// TIA Portal V20 export
FUNCTION_BLOCK "LER_hotPressLeftHistory"   // FB75, LAD
// stored: Access Published, MemoryReserve 100, SetENOAutomatically false
   VAR_INPUT
      finished : Bool;
      partID : String[32];
      ProductionTimestamp : DTL;
      result : Bool;
   END_VAR
   VAR_IN_OUT
      dataLog : "LER_typeServoPressHistory";
   END_VAR
   VAR
      statDataLogDelete { S7_SetPoint := 'True'} : "LER_typeServoPressHistory";
      statHold { S7_SetPoint := 'True'} : Bool;
      statExecute { S7_SetPoint := 'True'} : Bool;
      statMoveDone : Bool;
      statComplete { S7_SetPoint := 'True'} : Bool;
   END_VAR
   VAR_TEMP
      tempRetVal : Array[0..9] of Int;
      tempTrigger : Bool;
   END_VAR
   VAR_TEMP   // added for the SCL form of the ladder/FBD networks
      _w1 : Bool;
   END_VAR
BEGIN

REGION Network 1
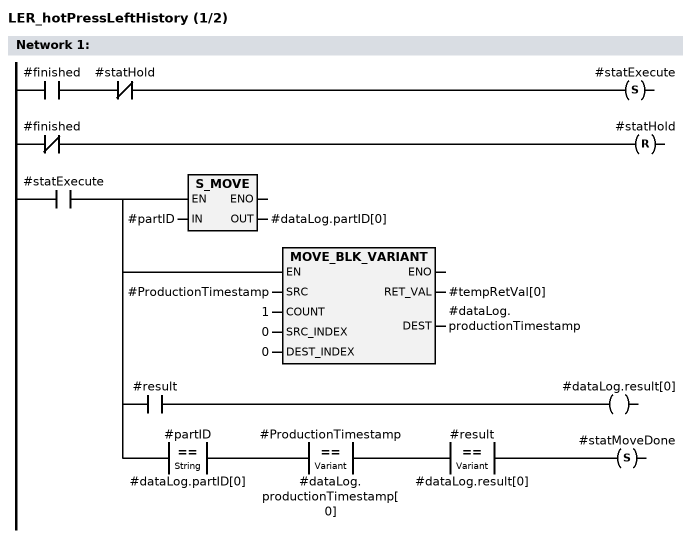
   RUNG wire#powerrail
      Contact( #finished )
      I_Contact( #statHold )
      S_Coil( #statExecute )
   END_RUNG
   RUNG wire#powerrail
      I_Contact( #finished )
      R_Coil( #statHold )
   END_RUNG
   RUNG wire#powerrail
      Contact( #statExecute )
      wire#w1
      S_Move(in := #partID, out => #dataLog.partID[0])
   END_RUNG
   RUNG wire#w1
      MOVE_BLK_VARIANT(SRC := #ProductionTimestamp, COUNT := 1, SRC_INDEX := 0, DEST_INDEX := 0, Ret_Val => #tempRetVal[0], DEST => #dataLog.productionTimestamp)
   END_RUNG
   RUNG wire#w1
      Contact( #result )
      Coil( #dataLog.result[0] )
   END_RUNG
   RUNG wire#w1
      { S7_Templates := "SrcType := String" } EQ_Contact(in1 := #partID, in2 := #dataLog.partID[0])
      { S7_Templates := "SrcType := Variant" } EQ_Contact(in1 := #ProductionTimestamp, in2 := #dataLog.productionTimestamp[0])
      { S7_Templates := "SrcType := Variant" } EQ_Contact(in1 := #result, in2 := #dataLog.result[0])
      S_Coil( #statMoveDone )
   END_RUNG
   // the same network as SCL:
   IF #finished AND NOT #statHold THEN #statExecute := TRUE; END_IF;
   IF NOT #finished THEN #statHold := FALSE; END_IF;
   IF #statExecute THEN
       #dataLog.partID[0] := #partID;
       #tempRetVal[0] := MOVE_BLK_VARIANT(SRC := #ProductionTimestamp,
                               COUNT := 1,
                               SRC_INDEX := 0,
                               DEST_INDEX := 0,
                               DEST => #dataLog.productionTimestamp);
   END_IF;
   #dataLog.result[0] := #statExecute AND #result;
   IF #statExecute AND (#partID = #dataLog.partID[0]) AND (#ProductionTimestamp = #dataLog.productionTimestamp[0]) AND (#result = #dataLog.result[0]) THEN
       #statMoveDone := TRUE;
   END_IF;
END_REGION

REGION Network 2
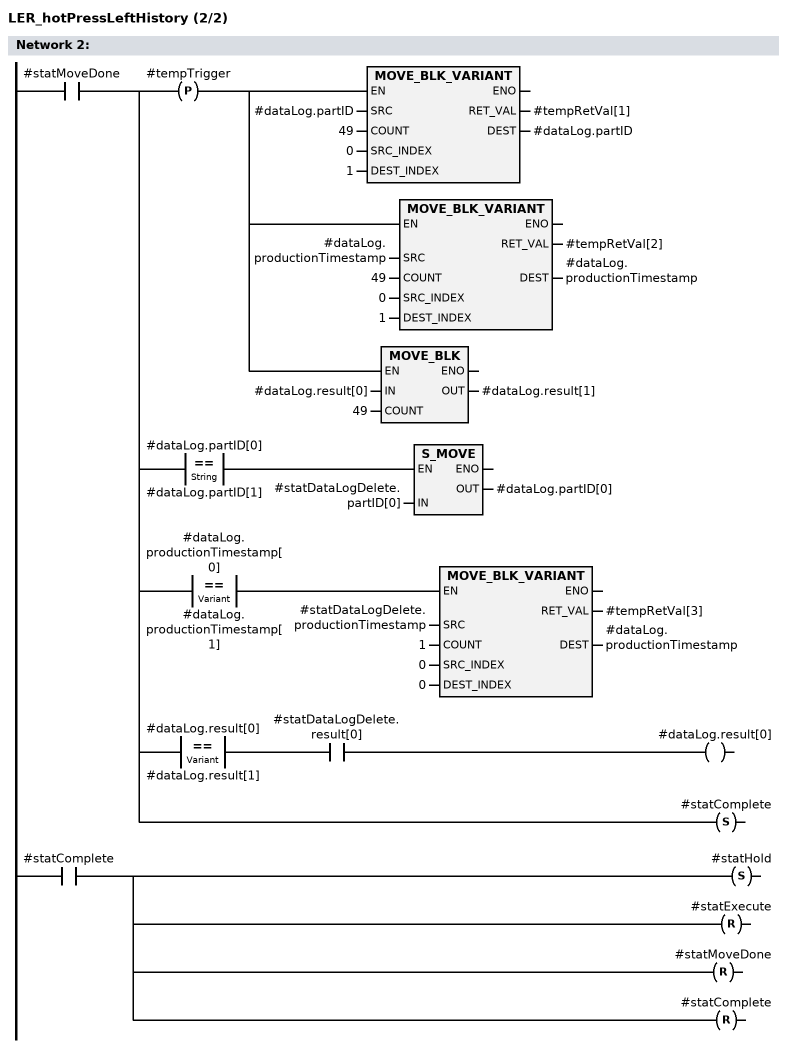
   #_w1 := #statMoveDone AND NOT #tempTrigger;   // rising edge
   #tempTrigger := #statMoveDone;
   IF #_w1 THEN
       #tempRetVal[1] := MOVE_BLK_VARIANT(SRC := #dataLog.partID,
                               COUNT := 49,
                               SRC_INDEX := 0,
                               DEST_INDEX := 1,
                               DEST => #dataLog.partID);
       #tempRetVal[2] := MOVE_BLK_VARIANT(SRC := #dataLog.productionTimestamp,
                               COUNT := 49,
                               SRC_INDEX := 0,
                               DEST_INDEX := 1,
                               DEST => #dataLog.productionTimestamp);
       MOVE_BLK(IN := #dataLog.result[0], COUNT := 49, OUT => #dataLog.result[1]);
   END_IF;
   IF #statMoveDone AND (#dataLog.partID[0] = #dataLog.partID[1]) THEN
       #dataLog.partID[0] := #statDataLogDelete.partID[0];
   END_IF;
   IF #statMoveDone AND (#dataLog.productionTimestamp[0] = #dataLog.productionTimestamp[1]) THEN
       #tempRetVal[3] := MOVE_BLK_VARIANT(SRC := #statDataLogDelete.productionTimestamp,
                               COUNT := 1,
                               SRC_INDEX := 0,
                               DEST_INDEX := 0,
                               DEST => #dataLog.productionTimestamp);
   END_IF;
   #dataLog.result[0] := #statMoveDone AND (#dataLog.result[0] = #dataLog.result[1]) AND #statDataLogDelete.result[0];
   IF #statMoveDone THEN #statComplete := TRUE; END_IF;
   IF #statComplete THEN
       #statHold := TRUE;
       #statExecute := FALSE;
       #statMoveDone := FALSE;
       #statComplete := FALSE;
   END_IF;
END_REGION
END_FUNCTION_BLOCK
